(* CoDeSys 2.3.9.22 project: pr3.pro *)
(* Libraries: Util.lib 18.5.10 15:14:28, STANDARD.LIB 4.10.05 11:14:46, IECSFC.LIB 13.4.06 15:51:28, ANALYZATION.LIB 5.10.99 09:05:06 *)

(* PLC configuration (modules and I/O channels)
PLC 150 I [Root] node -1, in %IB0 out %QB0 {MinCycleLength = 1; MaxCycleLength = 1000}
  Discrete input 6 bit [ID100] node 0, in %IB0 out %QB0 {Filtrationtime = 10; Filtrationtime = 10; Filtrationtime = 10; Filtrationtime = 10; Filtrationtime = 10; Filtrationtime = 10; Visibility = No; PinCount = 6; WatchDogPeriod = 1000; PollPeriod = 1}
    AT %IX0.0 [BitInput]
    AT %IX0.1 [BitInput]
    AT %IX0.2 [BitInput]
    AT %IX0.3 [BitInput]
    AT %IX0.4 [BitInput]
    AT %IX0.5 [BitInput]
  Discrete output 4 bit [ID101] node 1, in %IB1 out %QB1 {PinCount = 4; SafeValueBool = FALSE; SafeValueBool = FALSE; SafeValueBool = FALSE; SafeValueBool = FALSE; Visibility = No}
    AT %QX1.0 [BitOutput]
    AT %QX1.1 [BitOutput]
    AT %QX1.2 [BitOutput]
    AT %QX1.3 [BitOutput]
  Special output [ID104] node 2, in %IB2 out %QB2 {Visibility = No; PinCount = 1}
    AT %QX2.0 [BitOutput] Special output
  Unifed signal sensor [ID700] node 3, in %IB3 out %QB3 {Type_of_sensor700 = IT_0_20; measure_interval = 0.8; ainlow = 0; ainhigh = 20; first_cor_point = 0; first_delta = 0; second_cor_point = 0; second_delta = 0; third_cor_point = 0; third_delta = 0; Visibility = No}
    AT %ID3.0 [FloatInput] Value
    AT %IW3.1 [WordInput] Circular time
    Analog Input [ID107] node 0, in %IB3.0 out %QB3.0
  Unifed signal sensor [ID700] node 4, in %IB4 out %QB4 {Type_of_sensor700 = IT_0_20; measure_interval = 0.8; ainlow = 0; ainhigh = 20; first_cor_point = 0; first_delta = 0; second_cor_point = 0; second_delta = 0; third_cor_point = 0; third_delta = 0; Visibility = No}
    AT %ID4.0 [FloatInput] Value
    AT %IW4.1 [WordInput] Circular time
    Analog Input [ID107] node 0, in %IB4.0 out %QB4.0
  Unifed signal sensor [ID700] node 5, in %IB5 out %QB5 {Type_of_sensor700 = IT_0_20; measure_interval = 0.8; ainlow = 0; ainhigh = 20; first_cor_point = 0; first_delta = 0; second_cor_point = 0; second_delta = 0; third_cor_point = 0; third_delta = 0; Visibility = No}
    AT %ID5.0 [FloatInput] Value
    AT %IW5.1 [WordInput] Circular time
    Analog Input [ID107] node 0, in %IB5.0 out %QB5.0
  Unifed signal sensor [ID700] node 6, in %IB6 out %QB6 {Type_of_sensor700 = IT_0_20; measure_interval = 0.8; ainlow = 0; ainhigh = 20; first_cor_point = 0; first_delta = 0; second_cor_point = 0; second_delta = 0; third_cor_point = 0; third_delta = 0; Visibility = No}
    AT %ID6.0 [FloatInput] Value
    AT %IW6.1 [WordInput] Circular time
    Analog Input [ID107] node 0, in %IB6.0 out %QB6.0
  Analog output [ID106] node 7, in %IB7 out %QB7 {DAC_Type = Current 4-20mA; Analog_offset_correction = 0; Analog_full_range_correction = 0; SafeValueFloat = 0; Visibility = No}
    AT %QD7.0 [FloatOutput] Value
  Analog output [ID106] node 8, in %IB8 out %QB8 {DAC_Type = Current 4-20mA; Analog_offset_correction = 0; Analog_full_range_correction = 0; SafeValueFloat = 0; Visibility = No}
    AT %QD8.0 [FloatOutput] Value
*)

(* POU PLC_PRG, CFC *)
PROGRAM PLC_PRG
VAR
	pusk: BOOL;
	rs_pusk: RS;
	pulse_gen: BLINK;
	ctu1: CTU;
	X: REAL;
	Y: REAL;
	test: BOOL;
	ctu_isOdd: CTU;
	ton1: TON;
	ctu2: CTU;
	rs1: RS;
	power: BOOL;
	ctu3: CTU;
	ton2: TON;
	a: WORD;
	rs2: RS;
	ctu4: CTU;
	ton4: TON;
	P2: BOOL;
	P7: BOOL;
	P4: BOOL;
	KB: BOOL;
	stop: BOOL;
	off: BOOL;
	even: BOOL;
	odd: BOOL;
	ctu5: CTU;
	up: BOOL;
	checkUp: BOOL;
END_VAR
_CFC_ (* Continuous Function Chart, elements in execution order *)
#0 even <= #2
#1 ctu_isOdd:CTU(CU: pusk, RESET: -, PV: -)
#2 EQ(#3, 0)
#3 MOD(#1.CV, 2)
#4 R off <= pusk
#5 S power <= pusk
#6 WORD_TO_BOOL(#3)
#7 pulse_gen:blink(ENABLE: power, TIMELOW: t#1ms, TIMEHIGH: t#1ms)
#8 AND(#6, #7.OUT, NOT #19.Q1)
#9 AND(#8, NOT #10.Q, #46.Q)
#10 ctu1:CTU(CU: #9, RESET: #18.Q, PV: 70)
#11 WORD_TO_REAL(#10.CV)
#12 MUL(#11, -1)
#13 ton1:TON(IN: #10.Q, PT: t#2s)
#14 AND(#15, power)
#15 EQ(X, -70)
#16 P2 <= #14
#17 AND(#13.Q, #8, NOT #18.Q, #46.Q)
#18 ctu2:CTU(CU: #17, RESET: #18.Q, PV: 70)
#19 rs1:RS(SET: #18.Q, RESET1: NOT #6)
#20 WORD_TO_REAL(#18.CV)
#21 R power <= stop
#22 rs2:RS(SET: #18.Q, RESET1: #32.Q)
#23 AND(#22.Q1, NOT #6, #7.OUT, NOT #24.Q, NOT #32.Q, #46.Q)
#24 ctu3:CTU(CU: #23, RESET: #32.Q, PV: 70)
#25 WORD_TO_REAL(#24.CV)
#26 ADD(#12, #20, #25, #34)
#27 X <= #26
#28 S off <= stop
#29 ton2:TON(IN: #24.Q, PT: T#3s)
#30 AND(NOT #22.Q1, NOT #24.Q)
#31 AND(#29.Q, #7.OUT, NOT #32.Q, #24.Q, #22.Q1, #46.Q)
#32 ctu4:CTU(CU: #31, RESET: #30, PV: 70)
#33 WORD_TO_REAL(#32.CV)
#34 MUL(#33, -1)
#35 EQ(X, 70)
#36 P7 <= #42
#37 Y <= #49
#38 EQ(X, 0)
#39 P4 <= #43
#40 odd <= #41
#41 EQ(#3, 1)
#42 AND(#35, power)
#43 AND(#38, power)
#44 KB <= #47
#45 AND(#7.OUT, up, NOT #46.Q)
#46 ctu5:CTU(CU: #45, RESET: -, PV: 20)
#47 EQ(-20, Y)
#48 WORD_TO_REAL(#46.CV)
#49 MUL(#48, -1)
#50 S power <= up
_END_CFC_
END_PROGRAM

(* Visualisation v1
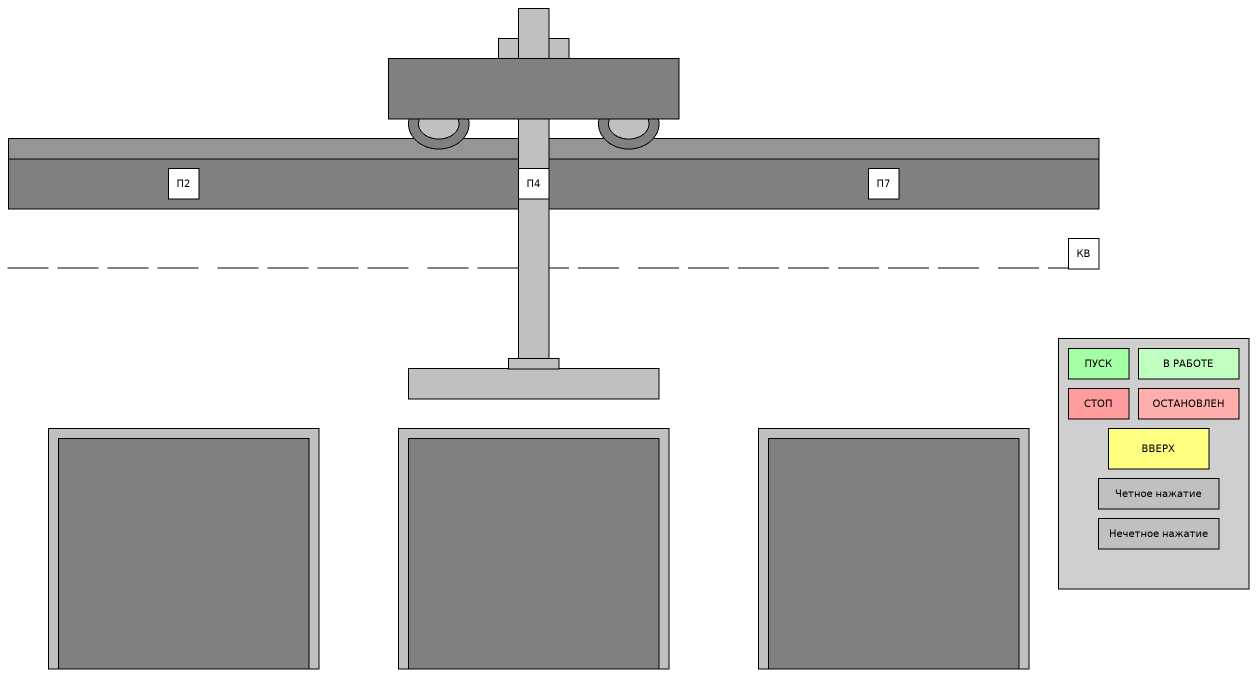
rounded rectangle at (1180,240)-(1241,271): text "ПУСК"; alarm colour if PLC_PRG.pusk; taps PLC_PRG.pusk
rounded rectangle at (1250,240)-(1351,271): text "В РАБОТЕ"; alarm colour if PLC_PRG.power
rounded rectangle at (1180,280)-(1241,311): text "СТОП"; alarm colour if PLC_PRG.stop; taps PLC_PRG.stop
rounded rectangle at (1250,280)-(1351,311): text "ОСТАНОВЛЕН"; alarm colour if PLC_PRG.off
rounded rectangle at (1210,370)-(1331,401): text "Четное нажатие"; alarm colour if PLC_PRG.even
rounded rectangle at (1210,410)-(1331,441): text "Нечетное нажатие"; alarm colour if PLC_PRG.odd
rectangle at (1180,130)-(1211,161): text "КВ"; alarm colour if PLC_PRG.KB
rounded rectangle at (610,-70)-(681,-49): x offset PLC_PRG.X*5
rectangle at (630,60)-(661,91): text "П4"; alarm colour if PLC_PRG.P4
rectangle at (280,60)-(311,91): text "П2"; alarm colour if PLC_PRG.P2
rectangle at (980,60)-(1011,91): text "П7"; alarm colour if PLC_PRG.P7
rounded rectangle at (1220,320)-(1321,361): text "ВВЕРХ"; alarm colour if PLC_PRG.up; taps PLC_PRG.up
38 more shapes without text or variables
*)
